Fanuc KAREL source: compact_preamble.KL

PROGRAM KT00094
%NOLOCKGROUP
VAR
H1 : ARRAY[2] OF SHORT
Y2 : ARRAY[2] OF BYTE
OUT:REAL
BEGIN
H1[1]=2
Y2[1]=3
OUT=((H1[1] * Y2[1]))
END KT00094
